FUNCTION_BLOCK XtsMoverTestSuite EXTENDS XtsMoverAxis
VAR
	fbTestSuites : FB_Testsuites;
	fbTestSuite : FB_Testsuite;
END_VAR

fbTestSuite();

CASE fbTestSuite.P_Testcase OF
	E_Testcase.Start:
		THIS^._MyNCData.AxisId := 1;
		fbTestSuite.P_Assert.M_Equals_DINT(1, THIS^.Cycle(), 'Cycle method did not return a complete');
		fbTestSuite.M_Testcase('GivenTheMoverIsFoundWhenCycleCalledThenCyclicTaskShouldRun',T#1S,'','',1);
		
	1:
		THIS^._MyNCData.AxisId := 0;
		fbTestSuite.P_Assert.M_Equals_DINT(-1, THIS^.Cycle(), 'Cycle method ran without vaild NC connection');
		fbTestSuite.M_Testcase('GivenNoNCWhenCycleCalledThenCyclicShouldNotRun',T#1S,'','',2);	
		
	2:
		_MyAxisStatus.Disabled := TRUE;
		fbTestSuite.P_Assert.M_Equals_DINT(1, THIS^.EnableMover(), 'Enable command failed when mover disabled');
		fbTestSuite.M_Testcase('GivenMoverDisabledWhenEnableCommandThenMoverEnables',T#1S,'','',3);
		
	3:
		_MyAxisStatus.Disabled := FALSE;
		fbTestSuite.P_Assert.M_Equals_DINT(-1, THIS^.EnableMover(), 'Enable Command was accepted when enabled');
		fbTestSuite.M_Testcase('GivenMoverEnabledWhenEnableComandThenEnableRejected',T#1S,'','',4);
		
	4:
		_MyAxisStatus.Disabled := FALSE;
		fbTestSuite.P_Assert.M_Equals_DINT(1, THIS^.DisableMover(), 'Disable command failed when mover was enabled');
		fbTestSuite.M_Testcase('GivenMoverEnabledWhenDisabledCommandMadeThenMoverDisables',T#1S,'','',5);
		
	5:	
		_MyAxisStatus.Disabled := TRUE;
		fbTestSuite.P_Assert.M_Equals_DINT(-1, THIS^.DisableMover(), 'Disable command accepted when mover was disabled');
		fbTestSuite.M_Testcase('GivenMoverDisabledWhenDisabledCommandMadeThenDisableRejected',T#1S,'','',6);
		
	6:
		_ActiveTrackLength := 5000.0;
		fbTestSuite.P_Assert.M_Equals_DINT(1,THIS^.MoveTo(RequiredPosition := 1000.0, MoveVelocity := 1000.0), 'Move command was rejected when mover was ready');
		fbTestSuite.M_Testcase('GivenMoverReadyWhenMoveCommandMadeThenMoverShouldAcceptMove',T#1S,'','',7);
		
	7:
		fbTestSuite.P_Assert.M_Equals_DINT(-1,THIS^.MoveTo(RequiredPosition := 1000.0, MoveVelocity := 5000.0), 'Move command was accepted when velocity too high');
		fbTestSuite.M_Testcase('WhenMoveCommandVelocityTooHighThenMoverShouldRejectMove',T#1S,'','',8);
		
	8: 
		_ActiveTrackLength := 1500.0;
		fbTestSuite.P_Assert.M_Equals_DINT(-1,THIS^.MoveTo(RequiredPosition := 2000.0, MoveVelocity := 1000.0), 'Move command was accepted when position outside modulo');
		fbTestSuite.M_Testcase('WhenMoveCommandOutsideModuloThenMoverShouldRejectMove',T#1S,'','',9);
		
	9:
		THIS^._MyAxisStatus.NotMoving := FALSE;
		fbTestSuite.P_Assert.M_Equals_DINT(1,THIS^.HaltAxis(),'Mover halt was rejected when mover moving');
		fbTestSuite.M_Testcase('GivenMovingMoverWhenHaltCommandThenMoverShouldAcceptHalt',T#1S,'','',10);
		
	10:
		THIS^._MyAxisStatus.NotMoving := FALSE;
		THIS^.HaltAxis();
		fbTestSuite.P_Assert.M_Equals_DINT(-1,THIS^.HaltAxis(), 'Mover halt was accepted when halt already commanded');
		fbTestSuite.M_Testcase('GivenHaltingMoverWhenHaltCommandGivenThenMoverShouldRejectCommand',T#1S,'','',11);
	
	11:
		THIS^.MoverHaltCommand.Abort();
		THIS^._MyAxisStatus.NotMoving := TRUE;
		fbTestSuite.P_Assert.M_Equals_DINT(-1,THIS^.HaltAxis(), 'Mover halt was accepted when velo was zero');
		fbTestSuite.M_Testcase('GivenStationaryMoverWhenHaltCommandedThenMoverShourlRejectCommand',T#1S,'','',12);
	
	12:
		THIS^.MoverResetCommand.Abort();
		THIS^._MyAxisStatus.Error := TRUE;
		fbTestSuite.P_Assert.M_Equals_DINT(1,THIS^.ResetAxis(), 'Mover reset was rejected when mover in error');
		fbTestSuite.M_Testcase('GivenMoverErrorWhenResetCommandedThemMoverShouldAcceptReset',T#1S,'','',13);
		
	13:
		THIS^._MyAxisStatus.Error := TRUE;
		THIS^.ResetAxis();
		fbTestSuite.P_Assert.M_Equals_DINT(-1,THIS^.ResetAxis(), 'Mover reset was accepted when reset already commanded');
		fbTestSuite.M_Testcase('GivenResettingMoverWhenResetCommandedThenMoverShouldRejectCommand',T#1S,'','',14);
		
	14:
		THIS^.MoverResetCommand.Abort();
		THIS^._MyAxisStatus.Error := FALSE;
		fbTestSuite.P_Assert.M_Equals_DINT(-1,THIS^.ResetAxis(), 'Mover reset was accepted when no error');
		fbTestSuite.M_Testcase('GivenOKMoverWhenResetCommandedThenMoverShouldRejectCommand',T#1S,'','',E_Testcase.Done);
		
	E_Testcase.Done:;	 
END_CASE

METHOD FB_init : BOOL
VAR_INPUT
	bInitRetains : BOOL; // if TRUE, the retain variables are initialized (warm start / cold start)
	bInCopyCode : BOOL;  // if TRUE, the instance afterwards gets moved into the copy code (online change)
END_VAR
//// Add Testsuite to Testsuites
TestSuiteGVL.fbTestsuites.M_Add(fbTestsuite);
TestSuiteGVL.fbTestsuites.P_Options.sFilePathName:= 'C:\test\report.xml';
END_METHOD

END_FUNCTION_BLOCK

(* stored: Version 1.1.0.1, ProductVersion 3.1.4024.12
   POU XtsMoverTestSuite: Id {0851a5af-3a91-4347-bf84-40e9438cdb23}, SpecialFunc None
   Method FB_init: Id {89d1ac51-1a68-4b8a-9c62-33c597fb6608} *)
